// TIA Portal V17 export
// export: Created 2023-02-13T11:16:52.6031479Z, ExportSetting WithDefaults, DisplayName Totally Integrated Automation Portal, DisplayVersion V17, DisplayName TIA Portal Openness, DisplayVersion V17, DisplayName TIA Portal Teamcenter Gateway, DisplayVersion V17, DisplayName TIA Portal Version Control Interface, DisplayVersion V17, DisplayName SINAMICS Startdrive Advanced, DisplayVersion V17, DisplayName SINAMICS Startdrive G130, G150, S120, S150, SINAMICS MV, S210, DisplayVersion V17, DisplayName SINAMICS Startdrive G110M, G120, G120C, G120D, G120P, G115D, DisplayVersion V17, DisplayName STEP 7 Professional, DisplayVersion V17, DisplayName STEP 7 Safety, DisplayVersion V17, DisplayName WinCC Professional, DisplayVersion V17
DATA_BLOCK "T-01.01_DB"   // DB351
VERSION : 0.1
// stored: AutoNumber false, DBAccessibleFromOPCUA true, DBAccessibleFromWebserver true, InstanceOfName HWT, InstanceOfType FB
"HWT"
   // VAR_INPUT
   //    "IN_FBAV.01" : Bool;
   //    "IN_FBAV.02" : Bool;
   //    "IN_FBAV.03" : Bool;
   //    "IN_FBAV.04" : Bool;
   //    "IN_FBAV.10" : Bool;
   //    "IN_FBCV.10" : Bool;
   //    "IN_FS.01" : Bool;
   //    IN_LT01 : Real;
   //    IN_TT01 : Real;
   //    IN_TT02 : Real;
   //    "IN_FBP.01" : Bool;
   //    "IN_P.01-Speed" : Real;
   //    DosePumpSpeed : Real;
   //    "DoseON-OFF" : Bool;
   //    "DosePumpON-OFF" : Bool;
   //    CIPPulse : Bool;
   //    Line_OK : Bool;
   // END_VAR
   // VAR_OUTPUT
   //    "OUT_AV.01" : Bool;
   //    "OUT_AV.02" : Bool;
   //    "OUT_AV.03" : Bool;
   //    "OUT_AV.04" : Bool;
   //    "OUT_AV.10" : Bool;
   //    "OUT_CV.10" : Bool;
   //    Q_PID_Setpoint : Real;
   //    Q_PID_PV_IN : Real;
   //    "OUT_FS.01" : Bool;
   //    "OUT_LT.01" : Real;
   //    "OUT_TT.01" : Real;
   //    "OUT_TT.02" : Real;
   //    "OUT_P.01" : Bool;
   //    "OUT_P.01-Speed" : Real;
   //    OUT_CIP_Request : Bool;
   //    Q_WH_Tank_Ready : Bool;
   // END_VAR
   // VAR
   //    Cmd : Struct
   //       Start_Prosses : Bool;
   //       Start_Preheat : Bool;
   //       HWT_Mode : Bool;
   //       Ready_for_Mix : Bool;
   //       "CIP Request" : Bool;
   //       Pump_Mode : Bool;
   //       Pump_Man_ON_OFF : Bool;
   //    END_STRUCT;
   //    Param : Struct
   //       SP_Level_LL : Real;
   //       SP_Level_ML : Real;
   //       SP_Level_HL : Real;
   //       SP_Temp_Prepar : Real;
   //       SP_Temp_Process : Real;
   //       SP_PumpSpeed : Real;
   //       L_Hi_Lim : Real;
   //       L_Lo_Lim : Real;
   //       L_Hys : Real;
   //       T_Hi_Lim : Real;
   //       T_Lo_Lim : Real;
   //       T_Hys : Real;
   //       CIP_Ret_ON_SP : Real;
   //       CIP_Ret_OFF_SP : Real;
   //    END_STRUCT;
   //    State : Struct
   //       Tank_LL : Bool;
   //       Tank_ML : Bool;
   //       Tank_HL : Bool;
   //       Temp_Preheat_OK : Bool;
   //       Temp_Process_OK : Bool;
   //       Tank_Heating : Bool;
   //       "Tank is Ready" : Bool;
   //       "Tank in transfer" : Bool;
   //       Enable_WHT_Mode : Bool;
   //       Enable_Ready : Bool;
   //       Ready_for_Mix : Bool;
   //       "CIP Request Enable" : Bool;
   //       "Tank in CIP" : Bool;
   //       CIP_Request_OK : Bool;
   //       CIP_ReturnON : Bool;
   //       HWT_Status : Int;
   //       Temp_Actual : Real;
   //    END_STRUCT;
   //    L_Hys_Abs : Real;
   //    T_Hys_Abs : Real;
   //    Hys_Level_HL : Real;
   //    Hys_Level_ML : Real;
   //    Hys_Level_LL : Real;
   //    "Hys SP_SP_Prepar" : Real;
   //    "Hys SP_SP_Process" : Real;
   //    "Hys SP_SP_" : Real;
   //    alwaysON : Bool;
   //    r : Struct
   //       PosE1 : Bool;
   //       PosE2 : Bool;
   //       PosE3 : Bool;
   //       PosE4 : Bool;
   //       PosE5 : Bool;
   //       PosE6 : Bool;
   //       PosE7 : Bool;
   //       PosE8 : Bool;
   //       PosE9 : Bool;
   //       PosE10 : Bool;
   //       PosE11 : Bool;
   //       PosE12 : Bool;
   //       PosE13 : Bool;
   //       PosE14 : Bool;
   //       PosE15 : Bool;
   //       PosE16 : Bool;
   //       PosE17 : Bool;
   //       PosE18 : Bool;
   //       PosE19 : Bool;
   //       PosE20 : Bool;
   //       PosE21 : Bool;
   //       PosE22 : Bool;
   //       PosE23 : Bool;
   //       PosE24 : Bool;
   //       PosE25 : Bool;
   //       PosE26 : Bool;
   //       PosE27 : Bool;
   //       PosE28 : Bool;
   //       PosE29 : Bool;
   //       PosE30 : Bool;
   //       PosE31 : Bool;
   //       PosE32 : Bool;
   //    END_STRUCT;
   //    Actuator : Struct
   //       AV_Inlet : Bool;
   //       AV_Return : Bool;
   //       CV_Steam : Bool;
   //       Pump : Bool;
   //    END_STRUCT;
   //    r_Pump : Bool;
   //    r_PumpTim { S7_SetPoint := 'True'} : IEC_TIMER;
   //    Alarm : Word;
   //    Event : Word;
   // END_VAR
BEGIN
END_DATA_BLOCK
